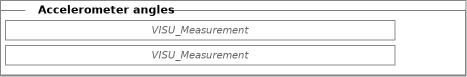
VISUALIZATION VISU_TelemetryAccelerometersAngles  // 467x77
VAR_IN_OUT
	ref : TelemetryAccelerometers;
    widget : TelemetryAccelerometersWidget;
END_VAR
    Polyline (170,10) (465,10) (465,75) (0,75) (0,10) (25,10)
    Label (35,0 140x20), "Accelerometer angles"
    Frame (5,20 390x20)
        shows VISU_Measurement(widget := widget.tubeX)
    Frame (5,45 390x20)
        shows VISU_Measurement(widget := widget.tubeY)
END_VISUALIZATION

(* stored: Version 1.1.0.1, ProductVersion 3.1.4019.2
   Visu VISU_TelemetryAccelerometersAngles: Id {9285dfb2-adfd-45ca-a3cd-32f72417bab6} *)
